// TIA Portal project "2-Motor Conveyor System" (V17)

(* hardware
DEVICE "S7-1200 station_1"  S7-1200 Station
   slot 0: "Rack_0"  S7-1200 Rack  Rack  V1.0
   slot 1: "PLC_1"  CPU 1214C DC/DC/DC  6ES7 214-1AG40-0XB0  V4.5
*)

// ===== PLC "PLC_1"  CPU 1214C DC/DC/DC =====

VAR_GLOBAL   // PLC tag table "Default tag table"
   "Start" AT %I0.0 : Bool;
   "Stop" AT %I0.1 : Bool;
   "Fault" AT %I0.2 : Bool;
   "Motor1_Run" AT %Q0.0 : Bool;
   "Object_detected" AT %I0.3 : Bool;
   "Motor2_Run" AT %Q0.1 : Bool;
   "Reset" AT %I0.4 : Bool;
   "Alarm" AT %Q0.2 : Bool;
END_VAR

DATA_BLOCK "Motor_1_DB"   // DB2
{ S7_Optimized_Access := 'TRUE' }
VERSION : 0.1
// stored: InstanceOfName Motor_1
"Motor_1"
BEGIN
END_DATA_BLOCK

DATA_BLOCK "Motor_2_DB"   // DB3
{ S7_Optimized_Access := 'TRUE' }
VERSION : 0.1
// stored: InstanceOfName Motor_2
"Motor_2"
BEGIN
END_DATA_BLOCK

DATA_BLOCK "Counter_DB"   // DB4
{ S7_Optimized_Access := 'TRUE' }
VERSION : 0.1
   VAR
      Object_counter : CTU_INT;
   END_VAR
BEGIN
END_DATA_BLOCK

// folder: System blocks/Program resources

DATA_BLOCK "Sort_timer_DB"   // DB1
{ S7_Optimized_Access := 'TRUE' }
AUTHOR : Simatic
FAMILY : IEC
NAME : IEC_TMR
VERSION : 1.0
// stored: InstanceOfName IEC_TIMER
"IEC_TIMER"
BEGIN
END_DATA_BLOCK

// folder: (top level)

FUNCTION_BLOCK "Motor_1"   // FB1, LAD
{ S7_Optimized_Access := 'TRUE' }
VERSION : 0.1
   VAR_INPUT
      Start : Bool;
      Stop : Bool;
      Fault : Bool;
   END_VAR
   VAR_OUTPUT
      Motor_Run : Bool;
   END_VAR
   VAR
      Latch : Bool;
   END_VAR
BEGIN

REGION Network 1
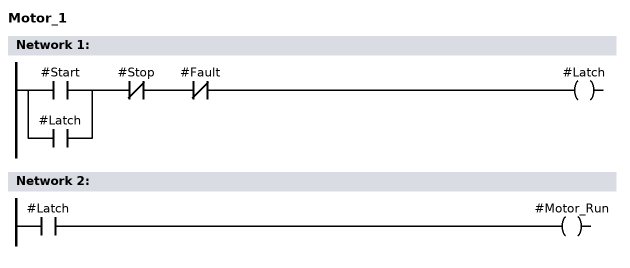
   RUNG wire#powerrail
      Contact( #Start )
      wire#w1
      I_Contact( #Stop )
      I_Contact( #Fault )
      Coil( #Latch )
   END_RUNG
   RUNG wire#powerrail
      Contact( #Latch )
   END_RUNG wire#w1
   // the same network as SCL:
   #Latch := (#Start OR #Latch) AND NOT #Stop AND NOT #Fault;
END_REGION

REGION Network 2
   RUNG wire#powerrail
      Contact( #Latch )
      Coil( #Motor_Run )
   END_RUNG
   // the same network as SCL:
   #Motor_Run := #Latch;
END_REGION
END_FUNCTION_BLOCK

FUNCTION_BLOCK "Motor_2"   // FB2, LAD
{ S7_Optimized_Access := 'TRUE' }
VERSION : 0.1
   VAR_INPUT
      Object_Detechted : Bool;
      Motor1_running : Bool;
      Stop : Bool;
      Fault : Bool;
   END_VAR
   VAR_OUTPUT
      Motor2_run : Bool;
   END_VAR
   VAR
      Sort_timer : Bool;
   END_VAR
BEGIN

REGION Network 1
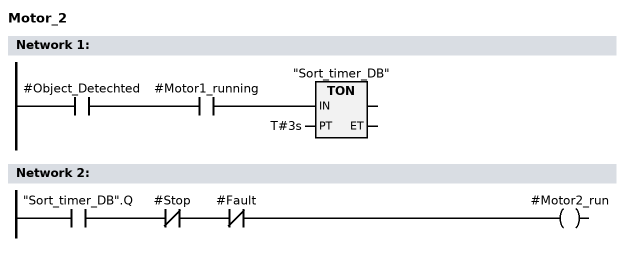
   "Sort_timer_DB".TON(IN := #Object_Detechted AND #Motor1_running, PT := T#3s);
END_REGION

REGION Network 2
   RUNG wire#powerrail
      Contact( "Sort_timer_DB".Q )
      I_Contact( #Stop )
      I_Contact( #Fault )
      Coil( #Motor2_run )
   END_RUNG
   // the same network as SCL:
   #Motor2_run := "Sort_timer_DB".Q AND NOT #Stop AND NOT #Fault;
END_REGION
END_FUNCTION_BLOCK

ORGANIZATION_BLOCK "Main"   // OB1, SCL, ProgramCycle
TITLE = "Main Program Sweep (Cycle)"
{ S7_Optimized_Access := 'TRUE' }
VERSION : 0.1
   VAR_INPUT
      Initial_Call : Bool;   // Initial call of this OB
      Remanence : Bool;   // =True, if remanent data are available
   END_VAR
BEGIN
   // ═══ MOTOR 1 — Main Conveyor Belt ═══
   "Motor_1_DB"(Start := "Start",
                Stop := "Stop",
                Fault := "Fault");

   "Motor1_Run" := "Motor_1_DB".Motor_Run;

   // ═══ MOTOR 2 — Sorting Arm ═══
   "Motor_2_DB"(Object_Detechted:="Object_detected",
                Motor1_running:="Motor_1_DB".Motor_Run,
                Stop:="Stop",
                Fault:="Fault");

   "Motor2_Run" := "Motor_2_DB".Motor2_run;

   // ═══ OBJECT COUNTER ═══
   "Counter_DB".Object_counter(
                               CU := "Object_detected",
                               R  := "Reset",
                               PV := 10);

   // ═══ AUTO STOP after 10 objects ═══
   IF "Counter_DB".Object_counter.QU THEN
       "Alarm" := TRUE; // Alarm light ON
   END_IF;

   IF "Reset" = TRUE THEN
       "Alarm" := FALSE;  // Reset alarm
   END_IF;
END_ORGANIZATION_BLOCK